FUNCTION_BLOCK T_ModuleCollectionInitialisedSuccess EXTENDS T_UnitTestBase
VAR
  list : T_SubModuleCollection(10);
  newModule, newModule2 : T_SubModuleMock; 
  actual1, actual2 : BOOL;
END_VAR

// Arrange
list.AddModule(newModule);
list.AddModule(newModule2);

//Act
list.CyclicLogic();

//Assert
actual1 := list.InitialisedAll;

assertion.AssertEquals_BOOL(TRUE, actual1, 'actual1 := list.InitialisedAll');
TestFinished();

END_FUNCTION_BLOCK

(* stored: Version 1.1.0.1, ProductVersion 3.1.4024.12
   POU T_ModuleCollectionInitialisedSuccess: Id {49bf7dae-95bb-46d1-be88-668cfa4a2532}, SpecialFunc None *)
